FUNCTION_BLOCK HandshakeResponderWSTRING (* Handshake pattern demo (WSTRING payload): Socket / Responder role *)
  (* Standard: 61499-2; Description: Copyright (c) 2026 Meisterschulen am Ostbahnhof This program and the accompanying materials are made available under the terms of the Eclipse Public License 2.0 which is available at https://www.eclipse.org/legal/epl-2.0/ SPDX-License-Identifier: EPL-2.0 *)
  (* Version 1.1, 2026-08-31, Franz Höpfinger, Meisterschulen am Ostbahnhof, HS.REQD/HS.CNFD/HS.INDD/HS.RSPD access syntax confirmed working in 4diac; ack payload moved to HandshakeConst::ACK_PAYLOAD (const/HandshakeConst.gcf) instead of a literal *)
  (* Version 1.0, 2026-08-31, Franz Höpfinger, Meisterschulen am Ostbahnhof, Handshake design pattern (IEC 61499 primer course, Module 6, Valeriy Vyatkin), demo Responder with WSTRING payload via EVENT_HS_WSTRING *)
  PACKAGE Meins::DesingPatterns::HandshakePattern;
  IMPORT Meins::DesingPatterns::HandshakePattern::const::HandshakeConst;
  (* Documentation:
  Responder ("server") side of the Handshake design pattern, data-carrying variant (IEC 61499 primer course, Module 6, Valeriy Vyatkin; adapter matches slide 48's generic "service" adapter).
   Uses adapter::events::Handshake::EVENT_HS_WSTRING as a Socket: receives REQ (reads HS.REQD into LastReqPayload) and answers with a fixed "ack" CNF; on TRIGGER it loads IndPayload into HS.INDD and sends an unsolicited IND; reads the matching RSP's payload into LastRspPayload.
   See HandshakePattern.md in this folder for the full write-up.
  *)
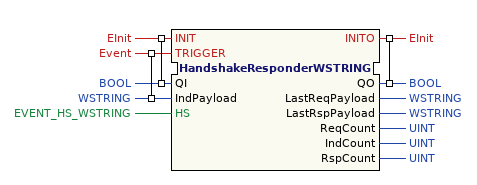
  EVENT_INPUT
    INIT : EInit WITH QI; (* Initialization Request *)
    TRIGGER WITH IndPayload; (* Demo: fire an unsolicited IND (with IndPayload) towards the Requester *)
  END_EVENT
  EVENT_OUTPUT
    INITO : EInit WITH QO; (* Initialization Confirm *)
  END_EVENT
  VAR_INPUT
    QI : BOOL; (* Input event qualifier *)
    IndPayload : WSTRING := "status,ok"; (* Payload sent with the next IND *)
  END_VAR
  VAR_OUTPUT
    QO : BOOL; (* Output event qualifier *)
    LastReqPayload : WSTRING; (* Payload of the last received REQ *)
    LastRspPayload : WSTRING; (* Payload of the last received RSP *)
    ReqCount : UINT; (* Number of REQ received (demo counter) *)
    IndCount : UINT; (* Number of IND sent (demo counter) *)
    RspCount : UINT; (* Number of RSP received (demo counter) *)
  END_VAR
  SOCKETS
    HS : adapter::types::bidirectional::Handshake::EVENT_HS_WSTRING; (* Handshake socket: receives REQ/RSP (+REQD/RSPD), emits CNF/IND (+CNFD/INDD) *)
  END_SOCKETS
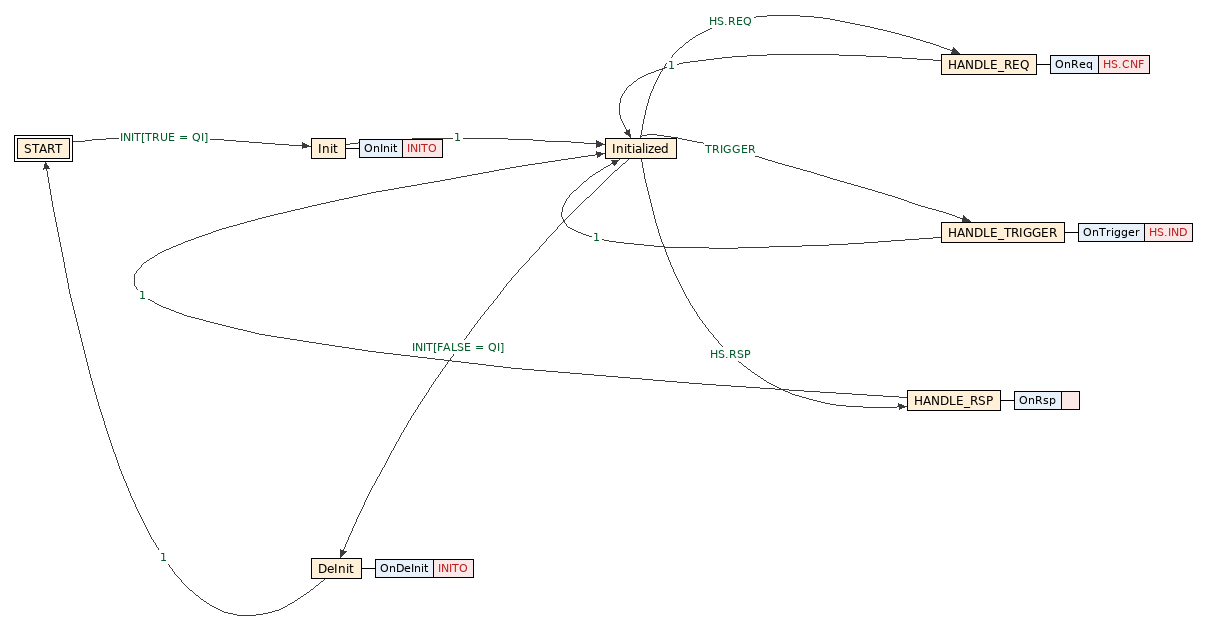
  EC_STATES
    START; (* Uninitialized *)
    Init : OnInit -> INITO; (* Initialization *)
    Initialized; (* Idle, ready to react *)
    DeInit : OnDeInit -> INITO; (* De-initialization *)
    HANDLE_REQ : OnReq -> HS.CNF; (* Read REQD, answer with a fixed CNFD *)
    HANDLE_TRIGGER : OnTrigger -> HS.IND; (* Load INDD from IndPayload, send an unsolicited IND *)
    HANDLE_RSP : OnRsp; (* Read RSPD, acknowledge an RSP *)
  END_STATES
  EC_TRANSITIONS
    START TO Init := INIT[TRUE = QI];
    Init TO Initialized := 1;
    Initialized TO DeInit := INIT[FALSE = QI];
    DeInit TO START := 1;
    Initialized TO HANDLE_REQ := HS.REQ;
    HANDLE_REQ TO Initialized := 1;
    Initialized TO HANDLE_TRIGGER := TRIGGER;
    HANDLE_TRIGGER TO Initialized := 1;
    Initialized TO HANDLE_RSP := HS.RSP;
    HANDLE_RSP TO Initialized := 1;
  END_TRANSITIONS
  ALGORITHM OnInit IN ST: (* Reset demo counters/payloads *)
ReqCount := 0;
IndCount := 0;
RspCount := 0;
LastReqPayload := "";
LastRspPayload := "";
QO := QI;
  END_ALGORITHM
  ALGORITHM OnDeInit IN ST: (* De-initialize *)
QO := FALSE;
  END_ALGORITHM
  ALGORITHM OnReq IN ST: (* Read REQD, count a received REQ, prepare a fixed CNFD *)
LastReqPayload := HS.REQD;
ReqCount := ReqCount + 1;
HS.CNFD := HandshakeConst::ACK_PAYLOAD;
  END_ALGORITHM
  ALGORITHM OnTrigger IN ST: (* Load INDD from IndPayload, count an IND about to be sent *)
HS.INDD := IndPayload;
IndCount := IndCount + 1;
  END_ALGORITHM
  ALGORITHM OnRsp IN ST: (* Read RSPD, count a received RSP *)
LastRspPayload := HS.RSPD;
RspCount := RspCount + 1;
  END_ALGORITHM
END_FUNCTION_BLOCK
